// TwinCAT 3 PLC project NewPLC
// ProgramVersion: 3.1.4023.0
// libraries:
//   Tc2_Standard, * (Beckhoff Automation GmbH)
//   Tc2_System, * (Beckhoff Automation GmbH)
//   Tc3_BA_Common, * (Beckhoff Automation GmbH)
//   Tc3_Module, * (Beckhoff Automation GmbH)
// project tree:
//   DUTs/Data Structures/ IntQueue.TcPOU
//   DUTs/Enumerations/Materials By Side/ BottomMaterialsEnum.TcTLEO, SidesMaterialsEnum.TcTLEO, TopMaterialsEnum.TcTLEO
//   DUTs/Enumerations/ EventsEnum.TcTLEO, AllMaterialsEnum.TcTLEO
//   DUTs/ MaterialPosition.TcDUT, PositionMaterials.TcDUT, PaperInterval.TcDUT
//   GVLs/ GVL.TcGVL
//   GVLs/Recipe/ BundleData.TcGVL, ExtrusionData.TcGVL, StrapWrapRecipe.TcGVL
//   / PlcTask.TcTTO
//   POUs/ AddRecipeToDatabase.TcPOU, MAIN.TcPOU, PrepareData.TcPOU
//   POUs/Functions/ ArrayContains.TcPOU, Control.TcPOU, SortMaterialPositionArray.TcPOU, SwapMaterialPosition.TcPOU
// real-time tasks:
//   TASK PlcTask: cycle T#10ms, priority 20, ADS port 350
//   TASK PlcTask1: cycle T#10ms, priority 21, ADS port 351
//   TASK PlcTask2: cycle T#10ms, priority 22, ADS port 352
//   TASK PlcTask3: cycle T#10ms, priority 23, ADS port 353
//   TASK PlcTask4: cycle T#10ms, priority 24, ADS port 354
//   TASK PlcTask5: cycle T#10ms, priority 25, ADS port 355

CONFIGURATION NewPLC
    RESOURCE PLC ON TwinCAT3
        TASK PlcTask(INTERVAL := T#10ms, PRIORITY := 21);
        PROGRAM MAIN WITH PlcTask : MAIN;
    END_RESOURCE
END_CONFIGURATION

// ---- DUTs/Enumerations/Materials By Side/BottomMaterialsEnum.TcTLEO
{attribute 'qualified_only'}
{attribute 'strict'}
{attribute 'to_string'}
TYPE BottomMaterialsEnum :
(

	//CARDBOARD
	CAR20S, CAR20M, CAR20L, CAR28S, CAR28M, CAR28L, //base (flat)
	
	//CHIPBOARD
	CIP18, CIP54,
	
	//WOOD BUNK
	WDB20, WDB22, WDB28, //bottom
	
	size //number of materials
);
END_TYPE

// ---- DUTs/Enumerations/Materials By Side/SidesMaterialsEnum.TcTLEO
{attribute 'qualified_only'}
{attribute 'strict'}
{attribute 'to_string'}
TYPE SidesMaterialsEnum :
(
	//CARDBOARD
	CAR20S, CAR20M, CAR20L, CAR28S, CAR28M, CAR28L, //base (flat)
	
	//CHIPBOARD
	CIP18, CIP54,
	
	//WOOD BUNK
	WDS08, WDS10, WDS12, WDS14, WDS20, WDS22, WDS28, //side
	WDS8X8, WDS8X10, WDS12X12, WDS12X14, WDS20X10, WDS20X12, //side combined - X
	
	size //number of materials
);
END_TYPE

// ---- DUTs/Enumerations/Materials By Side/TopMaterialsEnum.TcTLEO
{attribute 'qualified_only'}
{attribute 'strict'}
TYPE TopMaterialsEnum :
(
	//CARDBOARD
	CAR20S, CAR20M, CAR20L, CAR28S, CAR28M, CAR28L, //base (flat)
	
	//CHIPBOARD
	CIP18, CIP54,
	
	//WOOD BUNK
	WDT20, WDT22, WDT28, //top
	WDW20, WDW22, //special top (wide)
	
	size //number of materials
);
END_TYPE

// ---- DUTs/Enumerations/EventsEnum.TcTLEO
{attribute 'qualified_only'}
{attribute 'strict'}
//{attribute 'to_string'}
TYPE EventsEnum :
(
	//standard operation
	//BUNDLE_SENT, // = 0
	BUNDLE_RECEIVED,
	BUNDLE_COMPLETE,
	
	//area complete
	//AREA_1_COMPLETE,
	AREA_2_COMPLETE, //for this area
	//AREA_3_COMPLETE,
	//AREA_4_COMPLETE,
	//AREA_5_COMPLETE,
	//AREA_6_COMPLETE,
	
	//area specific operations
	SECTION_4_COMPLETE,
	SECTION_3_2_1_COMPLETE,
	SECTION_5_COMPLETE,
	SECTION_6_COMPLETE,

	//standard errors
	BACKLOG,
	MACHINE_FAILURE,
	DELAY,
	BUNDLE_EARLY_RECEIVED,
	BUNDLE_LATE_RECEIVED,
	
	//area specific errors
	SECTION_1_FAIL,
	SECTION_2_3_4_FAIL,
	SECTION_5_FAIL,
	SECTION_6_FAIL,
	
	//robots, motors, database, connections, etc
	
	size
);
END_TYPE

// ---- DUTs/Enumerations/AllMaterialsEnum.TcTLEO
{attribute 'qualified_only'}
{attribute 'strict'}
{attribute 'to_string'}
TYPE AllMaterialsEnum :
(
	//SIDES
	TOP, SIDES, BOTTOM,

	//CARDBOARD
	CAR20S, CAR20M, CAR20L, CAR28S, CAR28M, CAR28L, //base (flat)
	CAR20SF, CAR20MF, CAR20LF, CAR28SF, CAR28MF, CAR28LF, //single folded (L shape) - F
	CAR20SD, CAR20MD, CAR20LD, CAR28SD, CAR28MD, CAR28LD, //double folded (C shape) - D
	
	//CHIPBOARD
	CIP18, CIP54,
	
	//CORNER GUARD
	COR48,
	
	//PAPER
	PAP28,
	
	//WOOD BUNK
	WDT20, WDT22, WDT28, //top
	WDB20, WDB22, WDB28, //bottom
	WDS08, WDS10, WDS12, WDS14, WDS20, WDS22, WDS28, //side
	WDS8X8, WDS8X10, WDS12X12, WDS12X14, WDS20X10, WDS20X12, //side combined - X
	WDW20, WDW22, //special top (wide)
	
	size //number of materials
);
END_TYPE

// ---- DUTs/MaterialPosition.TcDUT
TYPE MaterialPosition :
STRUCT
	material : STRING;
	position : INT;
END_STRUCT
END_TYPE

// ---- DUTs/PositionMaterials.TcDUT
TYPE PositionMaterials :
STRUCT
	position : INT := 0; //default value is set to predefined constant if bundle needs less than 32 position material pairs
	
	//each position will only store 1 material per face
	top : STRING;
	sides : STRING;
	bottom : STRING;
	upperCorner : STRING;
	lowerCorner : STRING;
	
	wrap : BOOL; //for cardboard and corner guard only
END_STRUCT
END_TYPE

// ---- DUTs/PaperInterval.TcDUT
TYPE PaperInterval :
STRUCT
	start : INT;
	end : INT;
	
	wrap : BOOL;
END_STRUCT
END_TYPE

// ---- GVLs/GVL.TcGVL
{attribute 'qualified_only'}
{attribute 'global_init_slot' := '45000'}
VAR_GLOBAL CONSTANT //first to compile
	maxMaterials : INT := 13; //14-1
	maxPairs : INT := 24; //25-1
	
	top : ARRAY[1..TO_INT(TopMaterialsEnum.size)] OF STRING := [		'CAR20S', 'CAR20M', 'CAR20L', 'CAR28S', 'CAR28M', 'CAR28L', //CARDBOARD	
																		'CIP18', 'CIP54', //CHIPBOARD
																		'WDT20', 'WDT22', 'WDT28', 'WDW20', 'WDW22']; //WOOD BUNK
	
	sides : ARRAY[1..TO_INT(SidesMaterialsEnum.size)] OF STRING := [	'CAR20S', 'CAR20M', 'CAR20L', 'CAR28S', 'CAR28M', 'CAR28L', //CARDBOARD
																		'CIP18', 'CIP54', //CHIPBOARD
																		'WDS08', 'WDS10', 'WDS12', 'WDS14', 'WDS20','WDS22', 'WDS28', //WOOD BUNKS
																		'WDS8X8', 'WDS8X10', 'WDS12X12', 'WDS12X14', 'WDS20X10', 'WDS20X12'];
	
	bottom : ARRAY[1..TO_INT(BottomMaterialsEnum.size)] OF STRING := [	'CAR20S', 'CAR20M', 'CAR20L', 'CAR28S', 'CAR28M', 'CAR28L', //CARDBOARD
																		'CIP18', 'CIP54', //CHIPBOARD
																		'WDB20', 'WDB22', 'WDB28']; //WOOD BUNK
	
	//when inserted to database, materials here will be added to top and bottom materials
	upperCorner : ARRAY[1..8] OF STRING := ['COR48', //CORNER GUARD
											'CAR20SF', 'CAR20MF', 'CAR20LF', 'CAR28SF', 'CAR28MF', 'CAR28LF']; //CARDBOARD - SINGLE FOLDED
	lowerCorner : ARRAY[1..8] OF STRING := ['COR48', //CORNER GUARD
											'CAR20SF', 'CAR20MF', 'CAR20LF', 'CAR28SF', 'CAR28MF', 'CAR28LF']; //CARDBOARD - SINGLE FOLDED
	
	//by materials
	paper : ARRAY[0..0] OF STRING := ['PAP28'];
	cornerGuard : ARRAY[0..0] OF STRING := ['COR48'];
	
	cardboardTop : ARRAY[1..6] OF STRING := [	'CAR20S', 'CAR20M', 'CAR20L', 'CAR28S', 'CAR28M', 'CAR28L'];
	cardboardSides : ARRAY[1..6] OF STRING := [	'CAR20S', 'CAR20M', 'CAR20L', 'CAR28S', 'CAR28M', 'CAR28L'];
	cardboardBottom : ARRAY[1..6] OF STRING := [	'CAR20S', 'CAR20M', 'CAR20L', 'CAR28S', 'CAR28M', 'CAR28L'];
	cardboardUC : ARRAY[1..6] OF STRING := [	'CAR20SF', 'CAR20MF', 'CAR20LF', 'CAR28SF', 'CAR28MF', 'CAR28LF'];
	cardboardLC : ARRAY[1..6] OF STRING := [	'CAR20SF', 'CAR20MF', 'CAR20LF', 'CAR28SF', 'CAR28MF', 'CAR28LF'];
	
	chipboardTop : ARRAY[1..2] OF STRING := [	'CIP18', 'CIP54'];
	chipboardSides : ARRAY[1..2] OF STRING := [	'CIP18', 'CIP54'];
	chipboardBottom : ARRAY[1..2] OF STRING := ['CIP18', 'CIP54'];
	
	woodBunkTop : ARRAY[1..5] OF STRING := [	'WDT20', 'WDT22', 'WDT28', 'WDW20', 'WDW22'];
	woodBunkSides : ARRAY[1..13] OF STRING := [	'WDS08', 'WDS10', 'WDS12', 'WDS14', 'WDS20','WDS22', 'WDS28',
												'WDS8X8', 'WDS8X10', 'WDS12X12', 'WDS12X14', 'WDS20X10', 'WDS20X12'];										
	woodBunkBottom : ARRAY[1..3] OF STRING := [	'WDB20', 'WDB22', 'WDB28'];
END_VAR

// ---- GVLs/Recipe/BundleData.TcGVL
{attribute 'qualified_only'}
VAR_GLOBAL
	//HMI RECIPE
	id : STRING;
	weight : REAL;
	
	length : REAL;
	height : REAL;
	width : REAL;
	
	piecesHeight : USINT;
	piecesWidth : USINT;
	
	//processAreas : (AUTO_RE, MANUAL_RE, AUTO_SS, MANUAL_SS);
	requiredProcessing : ARRAY[0..3] OF BOOL;
	//IF AUTO_SS is selected then allow access to warp and strap recipe creation

END_VAR

// ---- GVLs/Recipe/ExtrusionData.TcGVL
{attribute 'qualified_only'}
VAR_GLOBAL	
	extrusionWeight : REAL;
	
	extrusionHeight : REAL;
	extrusionWidth : REAL;
END_VAR

// ---- GVLs/Recipe/StrapWrapRecipe.TcGVL
{attribute 'qualified_only'}
VAR_GLOBAL
	//v1 - entries are in the format of material-position separated by face
	TopMaterials : ARRAY[0..GVL.maxMaterials] OF MaterialPosition;
	SidesMaterials : ARRAY[0..GVL.maxMaterials] OF MaterialPosition;
	BottomMaterials : ARRAY[0..GVL.maxMaterials] OF MaterialPosition;

	UCMaterials : ARRAY[0..GVL.maxMaterials] OF MaterialPosition;
	LCMaterials : ARRAY[0..GVL.maxMaterials] OF MaterialPosition;
	
	//v2 - entries are in the format of position-material separated by material type
	faceCardboard : ARRAY[0..1] OF BOOL;
	facePaper : ARRAY[0..1] OF BOOL;
	
	TopPaper : ARRAY[0..4] OF PaperInterval;
	SidesPaper : ARRAY[0..4] OF PaperInterval;
	BottomPaper : ARRAY[0..4] OF PaperInterval;
	
	Cardboard : ARRAY[0..11] OF PositionMaterials;
	CornerGuard : ARRAY[0..4] OF PositionMaterials;
	
	Chipboard : ARRAY[0..7] OF PositionMaterials;
	WoodBunk : ARRAY[0..7] OF PositionMaterials;
	
	//plasticWrap : INT; //number of wrapping rotations at each position
END_VAR

// ---- POUs/MAIN.TcPOU
PROGRAM MAIN
VAR	
	generateRecipe : BOOL;
	
	prepareData : PrepareData;
	addRecipeToDB : AddRecipeToDatabase;
	
	launch : Control;
END_VAR

IF generateRecipe THEN
	prepareData();
	//addRecipeToDB();
END_IF

END_PROGRAM

// ---- POUs/PrepareData.TcPOU
FUNCTION_BLOCK PrepareData
VAR
	//local copy of StrapWrapRecipe arrays
	TopMaterials : ARRAY[0..GVL.maxMaterials] OF MaterialPosition;
	SidesMaterials : ARRAY[0..GVL.maxMaterials] OF MaterialPosition;
	BottomMaterials : ARRAY[0..GVL.maxMaterials] OF MaterialPosition;
	UCMaterials : ARRAY[0..GVL.maxMaterials] OF MaterialPosition;
	LCMaterials : ARRAY[0..GVL.maxMaterials] OF MaterialPosition;

	//database recipe
	paperArr : ARRAY[0..4] OF BOOL; //5 faces
	
	//array of structs
	cardboardArr : ARRAY[0..GVL.maxPairs] OF PositionMaterials;
	cornerGuardArr : ARRAY[0..GVL.maxPairs] OF PositionMaterials;
	chipboardArr : ARRAY[0..GVL.maxPairs] OF PositionMaterials;
	woodBunkArr : ARRAY[0..GVL.maxPairs] OF PositionMaterials;
	
	cardboardPositions : IntQueue;
	cornerGuardPositions : IntQueue;
	chipboardPositions : IntQueue;
	woodBunkPositions : IntQueue;
	
	allPositions : IntQueue;
	allPos : ARRAY[0..24] OF INT;
	
	step : (FETCH, ORGANIZE, COLLECT, CONVERT, GENERATE);
	manualLog : BOOL;
	
	i : INT;
END_VAR

CASE step OF
	FETCH: //put data into local data structures
		MEMCPY(ADR(TopMaterials), ADR(StrapWrapRecipe.TopMaterials), TO_UDINT(GVL.maxMaterials+1)*SIZEOF(MaterialPosition));
		MEMCPY(ADR(SidesMaterials), ADR(StrapWrapRecipe.SidesMaterials), TO_UDINT(GVL.maxMaterials+1)*SIZEOF(MaterialPosition));
		MEMCPY(ADR(BottomMaterials), ADR(StrapWrapRecipe.BottomMaterials), TO_UDINT(GVL.maxMaterials+1)*SIZEOF(MaterialPosition));
		MEMCPY(ADR(UCMaterials), ADR(StrapWrapRecipe.UCMaterials), TO_UDINT(GVL.maxMaterials+1)*SIZEOF(MaterialPosition));
		MEMCPY(ADR(LCMaterials), ADR(StrapWrapRecipe.LCMaterials), TO_UDINT(GVL.maxMaterials+1)*SIZEOF(MaterialPosition));
		
		cardboardPositions.clear();
		cornerGuardPositions.clear();
		chipboardPositions.clear();
		woodBunkPositions.clear();
		
	ORGANIZE:
		sort(TopMaterials);
		sort(SidesMaterials);
		sort(BottomMaterials);
		sort(UCMaterials);
		sort(LCMaterials);
	
	COLLECT:
		//iterate through face arrays to get positions for each material type
		collectMaterialPositions(cardboardPositions, 'CAR');
		collectMaterialPositions(cornerGuardPositions, 'COR');
		collectMaterialPositions(chipboardPositions, 'CIP');
		collectMaterialPositions(woodBunkPositions, 'WD');

		IF manualLog THEN
			FOR i:=0 TO allPositions.size()-1 BY 1 DO
				ADSLOGDINT(
					msgCtrlMask := ADSLOG_MSGTYPE_ERROR,
					msgFmtStr := 'allPositions.get() = %d',
					dintArg := allPositions.get(i));
			END_FOR
			manualLog := FALSE;
		END_IF
		
	CONVERT:
		//sort all positions
		cardboardPositions.sort();
		cornerGuardPositions.sort();
		chipboardPositions.sort();
		woodBunkPositions.sort();
		
		//NULL materials (material: '', position: -1) are all at the rear, all valid materials are at the front
		//we have all positions of each material type, now we iterate through those positions again and add materials to each pair
		convertToPositionMaterials();
		
	GENERATE:
		//log to database
		//refer to eventlogger sample
END_CASE

METHOD cleanup : BOOL //moves all NULL materials to the back
VAR_IN_OUT
	arr : ARRAY[*] OF MaterialPosition;
END_VAR
VAR
	//iterators
	i : INT;
END_VAR
(*
FOR i:=0 TO GVL.maxMaterials BY 1 DO
	IF arr[i].material = '' THEN //NULL material, shift elements forward
		MEMCPY(ADR(arr[i]), ADR(arr[i+1]), TO_INT(GVL.maxMaterials-i)*SIZEOF(MaterialPosition));
		arr[GVL.maxMaterials].material := '';
		arr[GVL.maxMaterials].position := -1;
	ELSE //valid material
		allPositions.offer(arr[i].position);
	END_IF
END_FOR
*)

FOR i:=GVL.maxMaterials TO 0 BY -1 DO //iterate backwards
	IF arr[i].material = '' THEN //NULL material, shift elements forward
		MEMCPY(ADR(arr[i]), ADR(arr[i+1]), TO_UDINT(GVL.maxMaterials-i)*SIZEOF(MaterialPosition));
		arr[GVL.maxMaterials].material := '';
		arr[GVL.maxMaterials].position := -1;
	ELSE //valid material
		allPositions.push(arr[i].position); //add position to arraylist
	END_IF
END_FOR
END_METHOD

METHOD collectMaterialPositions : BOOL
VAR_IN_OUT
	posQueue : IntQueue;
END_VAR
VAR_INPUT
	materialPrefix : STRING;
END_VAR
getAllPositionsFromFace(TopMaterials, posQueue, materialPrefix);
getAllPositionsFromFace(SidesMaterials, posQueue, materialPrefix);
getAllPositionsFromFace(BottomMaterials, posQueue, materialPrefix);
getAllPositionsFromFace(UCMaterials, posQueue, materialPrefix);;
getAllPositionsFromFace(LCMaterials, posQueue, materialPrefix);
END_METHOD

METHOD collectPositions_old : BOOL
VAR_IN_OUT
	arr : ARRAY[*] OF MaterialPosition;
END_VAR
VAR_INST
	//iterators
	i : INT;
END_VAR
FOR i:=0 TO GVL.maxMaterials BY 1 DO
	IF arr[i].material <> '' AND arr[i].position >= 0 THEN
		IF NOT allPositions.contains(arr[i].position) THEN //add new position if it does not exist yet
			allPositions.push(arr[i].position);
			ADSLOGDINT( //log
				msgCtrlMask := ADSLOG_MSGTYPE_ERROR, 
				msgFmtStr := 'New position found at iteration: %d',
				dintArg := i);
			ADSLOGDINT( //log
				msgCtrlMask := ADSLOG_MSGTYPE_ERROR, 
				msgFmtStr := 'Position: %d',
				dintArg := arr[i].position);
		END_IF
	END_IF
END_FOR
END_METHOD

METHOD convertToPositionMaterials : BOOL
VAR_INST
	i : INT;
END_VAR
FOR i:=0 TO allPositions.size()-1 BY 1 DO
	//find all cardboard from all sides with this position value 
	//nothing works here
	findMaterialsAtPosition(pair := cardboardArr[i], materialPrefix := 'CAR', position := allPositions.get(i));
	findMaterialsAtPosition(pair := cornerGuardArr[i], materialPrefix := 'COR', position := allPositions.get(i));
	findMaterialsAtPosition(pair := chipboardArr[i], materialPrefix := 'CIP', position := allPositions.get(i));
	findMaterialsAtPosition(pair := woodBunkArr[i], materialPrefix := 'WD', position := allPositions.get(i));
END_FOR
END_METHOD

METHOD findMaterialsAtPosition : BOOL
VAR_IN_OUT
	pair : PositionMaterials;
END_VAR
VAR_INPUT
	materialPrefix : STRING;
	position : INT;
END_VAR
VAR_INST
	i : INT;
END_VAR
pair.position := position;

//find 1 material for each face at this position
FOR i:=0 TO GVL.maxMaterials BY 1 DO
	IF FIND(StrapWrapRecipe.TopMaterials[i].material, materialPrefix) > 0 AND StrapWrapRecipe.TopMaterials[i].position = position THEN
		pair.top := StrapWrapRecipe.TopMaterials[i].material;
	END_IF
	IF FIND(StrapWrapRecipe.SidesMaterials[i].material, materialPrefix) > 0 AND StrapWrapRecipe.SidesMaterials[i].position = position THEN
		pair.sides := StrapWrapRecipe.SidesMaterials[i].material;
	END_IF
	IF FIND(StrapWrapRecipe.BottomMaterials[i].material, materialPrefix) > 0 AND StrapWrapRecipe.BottomMaterials[i].position = position THEN
		pair.bottom := StrapWrapRecipe.BottomMaterials[i].material;
	END_IF
	IF FIND(StrapWrapRecipe.UCMaterials[i].material, materialPrefix) > 0 AND StrapWrapRecipe.UCMaterials[i].position = position THEN
		pair.upperCorner := StrapWrapRecipe.UCMaterials[i].material;
	END_IF
	IF FIND(StrapWrapRecipe.LCMaterials[i].material, materialPrefix) > 0 AND StrapWrapRecipe.LCMaterials[i].position = position THEN
		pair.lowerCorner := StrapWrapRecipe.LCMaterials[i].material;
	END_IF
END_FOR
END_METHOD

METHOD findMaterialsAtPosition_1 : BOOL
VAR_IN_OUT
	pair : PositionMaterials;
	arr : ARRAY[*] OF MaterialPosition;
END_VAR
VAR_INPUT
	materialPrefix : STRING;
	position : INT;
END_VAR
VAR_INST
	i : INT; //iterator
	pairFaceNum : INT := 0;
END_VAR
pairFaceNum := 0;

pair.position := position;

//???
FOR i:=0 TO GVL.maxMaterials BY 1 DO
	IF FIND(arr[i].material, materialPrefix) > 0 AND arr[i].position = position THEN
		pair.top := arr[i].material;
		pairFaceNum := pairFaceNum + 1;
	END_IF
END_FOR
END_METHOD

METHOD getAllPositionsFromFace : BOOL
VAR_IN_OUT
	arr : ARRAY[*] OF MaterialPosition;
	posQueue : IntQueue;
END_VAR
VAR_INPUT
	//posQueue : IntQueue;
	materialPrefix : STRING;
END_VAR
VAR_INST
	//iterators
	i : INT;
END_VAR
FOR i:=0 TO GVL.maxMaterials BY 1 DO
	IF FIND(arr[i].material, materialPrefix) > 0 AND arr[i].position >= 0 THEN
		IF NOT posQueue.contains(arr[i].position) THEN
			posQueue.push(TopMaterials[i].position);
		END_IF
	END_IF
END_FOR
END_METHOD

METHOD pushToParallelArray : BOOL
VAR_IN_OUT
	destID : ARRAY[*] OF STRING;
	destPos : ARRAY[*] OF INT;
	
	src : ARRAY[*] OF MaterialPosition;
END_VAR
VAR_INST
	i : INT;
END_VAR
FOR i:=0 TO GVL.maxMaterials BY 1 DO
	destID[i] := src[i].material;
	destPos[i] := src[i].position;
END_FOR
END_METHOD

METHOD sort : BOOL //sorts array by position, uses bubblesort
VAR_IN_OUT
	arr : ARRAY[*] OF MaterialPosition;
END_VAR
VAR_INST
	//iterators
	i : INT;
	j : INT;
END_VAR
FOR i:=0 TO GVL.maxMaterials-1 BY 1 DO
	FOR j:=0 TO GVL.maxMaterials-i-1 BY 1 DO
		IF arr[j].material = '' THEN
			arr[j].position := -1;
			swap(arr[j], arr[j+1]);
		ELSIF arr[j].position > arr[j+1].position AND arr[j+1].material <> '' THEN
			swap(arr[j], arr[j+1]);
		END_IF
	END_FOR
END_FOR

(*
FOR i:=0 TO GVL.maxMaterials BY 1 DO
	IF arr[i].position >= 0 AND NOT allPositions.contains(arr[i].position) THEN
		allPositions.offer(arr[i].position); //add new position if it does not exist yet
		
		ADSLOGDINT( //log
			msgCtrlMask := ADSLOG_MSGTYPE_WARN, 
			msgFmtStr := 'Current iteration position: %d',
			dintArg := arr[i].position);
		
		ADSLOGDINT( //log
			msgCtrlMask := ADSLOG_MSGTYPE_ERROR, 
			msgFmtStr := 'New position found at iteration: %d',
			dintArg := i);
			
		ADSLOGDINT( //log
			msgCtrlMask := ADSLOG_MSGTYPE_ERROR, 
			msgFmtStr := 'New position value: %d',
			dintArg := arr[i].position);
	END_IF
END_FOR
*)
END_METHOD

METHOD sortParallelArrays : BOOL //sorts array by position, uses bubblesort
VAR_IN_OUT
	arrID : ARRAY[*] OF STRING;
	arrPos : ARRAY[*] OF INT;
END_VAR
VAR_INST
	//iterators
	i : INT;
	j : INT;
	
	tempID : STRING;
	tempPos : INT;
END_VAR
FOR i:=0 TO GVL.maxMaterials-1 BY 1 DO
	FOR j:=0 TO GVL.maxMaterials-i-1 BY 1 DO
		IF arrID[j] = '' THEN //swap anyways
			arrPos[j] := -1;
			
			//tempID := arrID[j];
			MEMCPY(ADR(tempID), ADR(arrID[j]), SIZEOF(STRING));
			tempPos := arrPos[j];
			
			//arrID[j] := arrID[j+1];
			MEMCPY(ADR(arrID[j]), ADR(arrID[j+1]), SIZEOF(STRING));
			arrPos[j] := arrPos[j+1];
			
			//arrID[j+1] := tempID;
			MEMCPY(ADR(arrID[j+1]), ADR(tempID), SIZEOF(STRING));
			arrPos[j+1] := tempPos;
		ELSIF arrPos[j] > arrPos[j+1] AND arrID[j+1] <> '' THEN //swap
			//tempID := arrID[j];
			MEMCPY(ADR(tempID), ADR(arrID[j]), SIZEOF(STRING));
			tempPos := arrPos[j];
			
			//arrID[j] := arrID[j+1];
			MEMCPY(ADR(arrID[j]), ADR(arrID[j+1]), SIZEOF(STRING));
			arrPos[j] := arrPos[j+1];
			
			//arrID[j+1] := tempID;
			MEMCPY(ADR(arrID[j+1]), ADR(tempID), SIZEOF(STRING));
			arrPos[j+1] := tempPos;
		END_IF
	END_FOR
END_FOR
END_METHOD

METHOD swap : BOOL
VAR_INPUT
	elem1 : REFERENCE TO MaterialPosition;
	elem2 : REFERENCE TO MaterialPosition;
END_VAR
VAR_INST
	temp : MaterialPosition;
END_VAR
//(*
MEMCPY(ADR(temp), ADR(elem1), SIZEOF(MaterialPosition)); //temp = arr[j]
MEMCPY(ADR(elem1), ADR(elem2), SIZEOF(MaterialPosition)); //arr[j] = arr[j+1]
MEMCPY(ADR(elem2), ADR(temp), SIZEOF(MaterialPosition)); //arr[j+1] = temp
//*)

(*
//temp = arr[j]
temp.material := elem1.material;
temp.position := elem1.position;

//arr[j] = arr[j+1]
elem1.material := elem2.material;
elem1.position := elem2.position;

//arr[j+1] = temp
elem2.material := temp.material;
elem2.position := temp.position;
*)
END_METHOD

END_FUNCTION_BLOCK

// ---- DUTs/Data Structures/IntQueue.TcPOU
FUNCTION_BLOCK IntQueue
VAR
	elements : FB_BA_DynamicArray := (uiEntrySize := SIZEOF(INT), uiMinExpCount := 4);
	length : USINT := 0;
END_VAR

METHOD clear : BOOL
VAR_INPUT
END_VAR
elements.Reset();
length := 0;
END_METHOD

METHOD contains : BOOL
VAR_INPUT
	value : INT;
END_VAR
VAR_INST
	i : INT;
END_VAR
IF length = 0 THEN
	contains := FALSE;
	RETURN;
END_IF

FOR i:=0 TO length-1 BY 1 DO
	IF get(i) = value THEN
		contains := TRUE;
		RETURN;
	END_IF
END_FOR
contains := FALSE;
END_METHOD

METHOD get : INT
VAR_INPUT
	i : INT;
END_VAR
elements.GetEntry(diIndex := i, pResultEntry := ADR(get));
END_METHOD

METHOD isEmpty : BOOL
VAR_INPUT
END_VAR
isEmpty := (length = 0);
END_METHOD

METHOD poll : INT
VAR_INST
	temp : INT;
	i : INT;
END_VAR
temp := get(i := 0);
elements.RemoveEntry(diIndex := 0);
length := length - 1;
poll := temp;
END_METHOD

METHOD push : BOOL
VAR_INPUT
	value : INT;
END_VAR
elements.AddEntry(pEntry := ADR(value));
length := length + 1;
END_METHOD

METHOD set : BOOL
VAR_INPUT
	i : INT;
	value : INT;
END_VAR
elements.SetEntry(i, ADR(value));
END_METHOD

METHOD size : USINT
VAR_INPUT
END_VAR
size := length;
END_METHOD

METHOD sort : BOOL
VAR_INPUT
END_VAR
VAR_INST
	i : INT;
	j : INT;
	temp : INT;
END_VAR
FOR i:=0 TO GVL.maxMaterials BY 1 DO
	FOR j:=0 TO GVL.maxMaterials BY 1 DO
		IF get(j) > get(j+1) THEN //swap
			temp := get(j);
			set(j, get(j+1));
			set(j+1, temp);
		END_IF
	END_FOR
END_FOR
END_METHOD

END_FUNCTION_BLOCK

// ---- POUs/AddRecipeToDatabase.TcPOU
FUNCTION_BLOCK AddRecipeToDatabase
VAR_INPUT
	//BundleData
	//ExtrusionData
	//StrapWrapRecipe
END_VAR
VAR
END_VAR

END_FUNCTION_BLOCK

// ---- POUs/Functions/Control.TcPOU
FUNCTION_BLOCK Control
VAR
	j : INT;
END_VAR

{attribute 'TcRpcEnable'}
METHOD removeBottomMaterial : BOOL
VAR_INPUT
	i : INT; //index to be removed
END_VAR
FOR j:=i TO GVL.maxMaterials-1 BY 1 DO
	MEMCPY(ADR(StrapWrapRecipe.bottomMaterials[j]), ADR(StrapWrapRecipe.bottomMaterials[j+1]), SIZEOF(MaterialPosition));
END_FOR

StrapWrapRecipe.bottomMaterials[GVL.maxMaterials].material := '';
StrapWrapRecipe.bottomMaterials[GVL.maxMaterials].position := 0;
END_METHOD

{attribute 'TcRpcEnable'}
METHOD removeLCMaterial : BOOL
VAR_INPUT
	i : INT; //index to be removed
END_VAR
FOR j:=i TO GVL.maxMaterials-1 BY 1 DO
	MEMCPY(ADR(StrapWrapRecipe.lcMaterials[j]), ADR(StrapWrapRecipe.lcMaterials[j+1]), SIZEOF(MaterialPosition));
END_FOR

StrapWrapRecipe.lcMaterials[GVL.maxMaterials].material := '';
StrapWrapRecipe.lcMaterials[GVL.maxMaterials].position := 0;
END_METHOD

{attribute 'TcRpcEnable'}
METHOD removeSidesMaterial : BOOL
VAR_INPUT
	i : INT; //index to be removed
END_VAR
FOR j:=i TO GVL.maxMaterials-1 BY 1 DO
	MEMCPY(ADR(StrapWrapRecipe.sidesMaterials[j]), ADR(StrapWrapRecipe.sidesMaterials[j+1]), SIZEOF(MaterialPosition));
END_FOR

StrapWrapRecipe.sidesMaterials[GVL.maxMaterials].material := '';
StrapWrapRecipe.sidesMaterials[GVL.maxMaterials].position := 0;
END_METHOD

{attribute 'TcRpcEnable'}
METHOD removeTopMaterial : BOOL
VAR_INPUT
	i : INT; //index to be removed
END_VAR
FOR j:=i TO GVL.maxMaterials-1 BY 1 DO
	MEMCPY(ADR(StrapWrapRecipe.topMaterials[j]), ADR(StrapWrapRecipe.topMaterials[j+1]), SIZEOF(MaterialPosition));
END_FOR

StrapWrapRecipe.topMaterials[GVL.maxMaterials].material := '';
StrapWrapRecipe.topMaterials[GVL.maxMaterials].position := 0;
END_METHOD

{attribute 'TcRpcEnable'}
METHOD removeUCMaterial : BOOL
VAR_INPUT
	i : INT; //index to be removed
END_VAR
FOR j:=i TO GVL.maxMaterials-1 BY 1 DO
	MEMCPY(ADR(StrapWrapRecipe.ucMaterials[j]), ADR(StrapWrapRecipe.ucMaterials[j+1]), SIZEOF(MaterialPosition));
END_FOR

StrapWrapRecipe.ucMaterials[GVL.maxMaterials].material := '';
StrapWrapRecipe.ucMaterials[GVL.maxMaterials].position := 0;
END_METHOD

END_FUNCTION_BLOCK

// ---- POUs/Functions/ArrayContains.TcPOU
FUNCTION ArrayContains : BOOL
VAR_IN_OUT
	arr : ARRAY[*] OF INT;
END_VAR
VAR_INPUT
	value : INT;
END_VAR
VAR
	i : DINT;
END_VAR

FOR i:=0 TO UPPER_BOUND(arr, 1) BY 1 DO
	IF arr[i] = value THEN
		ArrayContains := TRUE;
		RETURN;
	END_IF
END_FOR

ArrayContains := FALSE;

END_FUNCTION

// ---- POUs/Functions/SortMaterialPositionArray.TcPOU
FUNCTION SortMaterialPositionArray : BOOL
VAR_IN_OUT
	arr : ARRAY[*] OF MaterialPosition;
END_VAR
VAR
	//iterators
	i : INT;
	j : INT;
END_VAR

FOR i:=0 TO GVL.maxMaterials BY 1 DO
	FOR j:=0 TO GVL.maxMaterials BY 1 DO
		IF arr[j].position > arr[j+1].position THEN
			SwapMaterialPosition(ADR(arr[j]), ADR(arr[j+1]));
		END_IF
	END_FOR
END_FOR

END_FUNCTION

// ---- POUs/Functions/SwapMaterialPosition.TcPOU
FUNCTION SwapMaterialPosition : BOOL
VAR_INPUT
	elem1 : POINTER TO MaterialPosition;
	elem2 : POINTER TO MaterialPosition;
END_VAR
VAR
	temp : MaterialPosition;
END_VAR

MEMCPY(ADR(temp), elem1, SIZEOF(MaterialPosition)); //temp = arr[j]
MEMCPY(elem1, elem2, SIZEOF(MaterialPosition)); //arr[j] = arr[j+1]
MEMCPY(elem2, ADR(temp), SIZEOF(MaterialPosition)); //arr[j+1] = temp

END_FUNCTION
